TYPE ST_Results :
STRUCT
	tare: REAL;
	gross: REAL;
	rest: REAL;
	calibrationNo: INT;
	userId: STRING;
	density: REAL;
	solventNo: INT;
	solventRevision: INT;
	sysMasterRevision: INT;
	allowableFail: INT;
	replicates: INT;
	callInterval: INT;
	dateTime: STRING;
	pumpNo: INT;
	step: STRING;
	tareWt: REAL;
	grossWt: REAL;
	netVolume: REAL;
	netWt: REAL;
	targetVolume: REAL;
	differencePercent: REAL;
	criteria: REAL;
	pumpRevs: INT;
	Runs_ID: INT;
	
END_STRUCT
END_TYPE

(* stored: Version 1.1.0.1, ProductVersion 3.1.4024.12
   DUT ST_Results: Id {0a001843-8587-4884-94b6-5378f1bddf5e} *)
